Fanuc KAREL source: kt00206.KL

-- PROVISIONAL review KL for V1013-1; original PC SHA256 3c713106b7d1a9354bc3ecb726903d0dd5a5081acef8ce136aed6732459616c6
-- Incomplete behavior may be omitted. Consult companion uncertainty JSON. Do not deploy.
PROGRAM KT00206
%NOLOCKGROUP
VAR
  I1 : INTEGER
  OUT : INTEGER
-- UNRESOLVED_DECL Y2 type=002018
BEGIN
  -- UNRESOLVED_PC offsets 5-16; opcodes 2E,23
  -- UNRESOLVED_PC offsets 21-35; opcodes 2E,22,9D,33,B2
  -- UNRESOLVED_PC offsets 40-62; opcodes 21,22,9D,33,B1,46,23
  -- UNRESOLVED_PC offsets 67-71; opcodes 7F
END KT00206
